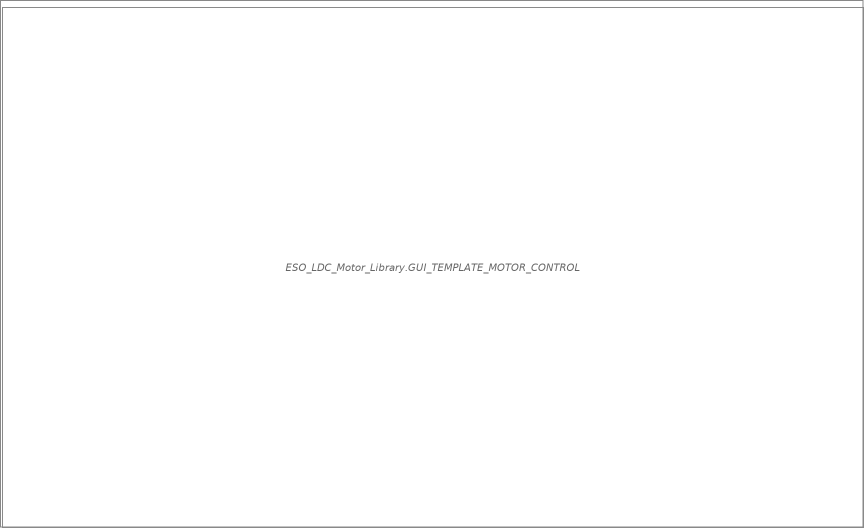
VISUALIZATION Motor001_Ctrl  // 864x528
    Frame (2,7 862x521)
        shows ESO_LDC_Motor_Library.GUI_TEMPLATE_MOTOR_CONTROL(m_Instance := MAIN.Motor001)
END_VISUALIZATION

(* stored: Version 1.1.0.1, ProductVersion 3.1.4024.9
   Visu Motor001_Ctrl: Id {8eefbd0a-d0ae-4311-910c-f485f00ee1ea} *)
